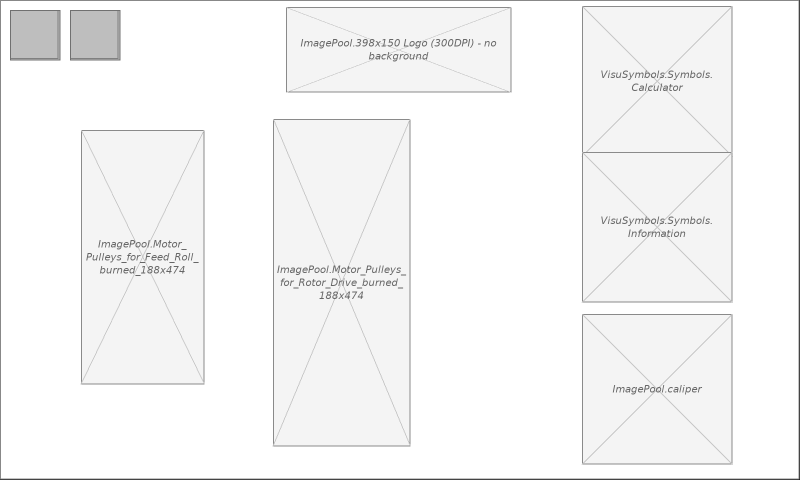
VISUALIZATION Settings_Menu  // 800x480
    Rectangle (0,0 800x480)
    Button (10,10 50x50), image: VisuSymbols.Symbols.TriangleLeft
        OnMouseClick: change screen: Previous Home
    Button (70,10 50x50), image: VisuSymbols.Symbols.Home
        OnMouseClick: change screen: Home
    Image (273,119 137x327), image: ImagePool.Motor_Pulleys_for_Rotor_Drive_burned_188x474
        OnMouseClick: change screen: Rotor_Settings
    Image (81,130 123x254), image: ImagePool.Motor_Pulleys_for_Feed_Roll_burned_188x474
        OnMouseClick: change screen: Feedroll_Settings
    Image (582,314 150x150), image: ImagePool.caliper
        OnMouseClick: change screen: Calibrate_Settings
    Image (582,6 150x150), image: VisuSymbols.Symbols.Calculator
        OnMouseClick: change screen: Calculations_Settings
    Image (582,152 150x150), image: VisuSymbols.Symbols.Information
        OnMouseClick: change screen: Machine_ID_Settings
    Image (286,7 225x85), image: ImagePool.398x150 Logo (300DPI) - no background
        OnMouseClick: change screen: Home
END_VISUALIZATION

(* stored: Version 1.1.0.1, ProductVersion 3.1.4024.12
   Visu Settings_Menu: Id {7a7b57fd-a097-4861-a13e-331f33588901} *)
